FUNCTION_BLOCK QualityInspectionContainer EXTENDS ZCore.ObjectContainer
VAR_INPUT
END_VAR
VAR_OUTPUT
END_VAR
VAR
  {attribute 'hide'}
  _parent : REFERENCE TO QualityInspectionUnit;
END_VAR

{ attribute 'hide' }
METHOD FB_init : BOOL
VAR_INPUT
	bInitRetains : BOOL; // if TRUE, the retain variables are initialized (warm start / cold start)
	bInCopyCode : BOOL;  // if TRUE, the instance afterwards gets moved into the copy code (online change)
  unit : REFERENCE TO QualityInspectionUnit;
END_VAR
_parent REF= unit;
END_METHOD

END_FUNCTION_BLOCK

(* stored: Version 1.1.0.1
   POU QualityInspectionContainer: Id {5c6f9e73-f785-41de-bf69-26011e2c00ab}, SpecialFunc None
   Method FB_init: Id {c132d320-529c-4e08-9ac9-b51e03fe004f} *)
